FUNCTION Convert_TOD_TO_DT : Hresult
VAR_INPUT
	in : TOD;
	out : REFERENCE TO DT;
END_VAR
VAR
	converted : DT;
END_VAR
VAR CONSTANT
	INCOMPATIBLE : HRESULT := 16#9811070E;
END_VAR

converted := TOD_TO_DT(in);

IF (DT_TO_TOD(converted) <> in) THEN
	Convert_TOD_TO_DT := INCOMPATIBLE;
	RETURN;
END_IF

out := converted;

END_FUNCTION

(* stored: Version 1.1.0.1, ProductVersion 3.1.4024.12
   POU Convert_TOD_TO_DT: Id {af379faf-eaee-4953-89ee-ec277123c165}, SpecialFunc None *)
